Universal Robots PolyScope program: 6 novembre.urp

Program 6 novembre (installation=default directory=/programs createdIn=3.15.8.106339 lastSavedIn=3.15.8.106339 robotSerialNumber=2023330214)
Calibrated DH parameters: a=[-0.000161, -0.243516, -0.175941, 0.000055, -0.000127, 0]; d=[0.151869, -0.926342, 57.568096, -56.529557, 0.085345, 0.082309]; alpha=[1.571543, -0.007517, 0.002128, 1.570286, -1.573097, 0]; deltaTheta=[0.000048, 0.028487, 0.571925, -0.600676, 0.000055, 0.000013]
BeforeStart
  conta := 0
Robot Program (runOnlyOnce=false)
  Loop Counting (count=5) loopVariable(name=Loop_1)
    MoveJ speed 60 deg/s, acceleration 80 deg/s^2 (useActiveTCP=true)
      Waypoint partenza: motionParameters(jointSpeed=6.283185 jointAcceleration=6.283185 cartesianSpeed=0.25 cartesianAcceleration=1.2); TCP in base x=295.823 y=29.54 z=245.993 mm, rx=-1.6446 ry=2.6015 rz=0.0088 rad; joints [31.55, -87.588, -89.18, -89.432, 90.433, 57.296] deg; flange x=307.635 y=60.145 z=330.959 mm, rx=-1.6446 ry=2.6015 rz=0.0088 rad
      Pallet pattern(dimensionality=Square firstAxisCount=2 secondAxisCount=2 thirdAxisCount=5 motionType=MoveL speed=0.25 acceleration=1.2 useActiveTCP=true, counterVariable(name=cnt_1, initializeExpression=0), patternPoseVariable(name=pose_1), feature=Base, children(Waypoint(type=Fixed name=Corner1_2, position(joints=1.7071903944015503, -2.0363944212542933, -1.974642578755514, -0.7177489439593714, 1.586946964263916, 1.8594038486480713 pose=0.05591609202787988, 0.3042326877636343, 0.04062971376229775, 2.037561659965045, -2.3576852381341817, 0.00967614852521311), poseInFeatureCoordinates=[0.055916, 0.304233, 0.04063, 2.037562, -2.357685, 0.009676], outputFlangePose=[0.062603, 0.343098, 0.122727, 2.037562, -2.357685, 0.009676]), Waypoint(type=Fixed name=Corner2_2, position(joints=1.3555443286895752, -2.164708439503805, -1.7350428740130823, -0.8342025915728968, 1.5785411596298218, 1.5071099996566772 pose=0.18014491122547477, 0.3042332340391118, 0.04060207246304333, 2.037508402011708, -2.357604882143758, 0.009722233499361176), poseInFeatureCoordinates=[0.180145, 0.304233, 0.040602, 2.037508, -2.357605, 0.009722], outputFlangePose=[0.186836, 0.343105, 0.122696, 2.037508, -2.357605, 0.009722]), Waypoint(type=Fixed name=Corner3_2, position(joints=1.2638148069381714, -1.8657797018634241, -2.2631152311908167, -0.6058977285968226, 1.5782291889190674, 1.4168099164962769 pose=0.18015284222828584, 0.1875657559943738, 0.04061133384541858, 2.03742066799229, -2.3576919944708794, 0.009735192963967047), poseInFeatureCoordinates=[0.180153, 0.187566, 0.040611, 2.037421, -2.357692, 0.009735], outputFlangePose=[0.186846, 0.226438, 0.122705, 2.037421, -2.357692, 0.009735]), Waypoint(type=Fixed name=Corner4_2, position(joints=1.8628913164138794, -1.6507962385760706, -2.576595131550924, -0.49827701250185186, 1.5922470092773438, 2.016301393508911 pose=0.03904266180606819, 0.18759146961099127, 0.040612373225184156, 2.0374934541390837, -2.3578468661229373, 0.009639408672472292), poseInFeatureCoordinates=[0.039043, 0.187591, 0.040612, 2.037493, -2.357847, 0.009639], outputFlangePose=[0.04573, 0.22645, 0.122713, 2.037493, -2.357847, 0.009639]))); actionSequence(name=PalletSequence motionType=MoveL speed=0.25 acceleration=1.2 useActiveTCP=true, anchorWaypoint(type=Fixed name=PatternPoint_2), feature=Base, children(Waypoint(type=Fixed name=Approach_2), Waypoint=PatternPoint_2, Set(type=Undefined), Wait(type=Undefined), Waypoint(type=Fixed name=Exit_2)))
        Pattern -> pattern
        AnchoredSequence -> PalletSequence
      Pallet pattern(dimensionality=Box firstAxisCount=2 secondAxisCount=2 thirdAxisCount=2 motionType=MoveL speed=2 acceleration=2 useActiveTCP=true, counterVariable(name=cnt_2, initializeExpression=0), patternPoseVariable(name=pose_2), feature=Base, children(Waypoint(type=Fixed name=Corner1_1, position(joints=1.5661438703536987, -2.322768513356344, -1.645829979573385, -0.6583693663226526, 1.5955449342727661, 0.8307483792304993 pose=0.13254062465471933, 0.3819871783574357, 0.01202495287692959, -2.815561845639961, 1.238537976676179, 0.09161537053473316), poseInFeatureCoordinates=[0.132541, 0.381987, 0.012025, -2.815562, 1.238538, 0.091615], outputFlangePose=[0.109614, 0.402639, 0.097717, -2.815562, 1.238538, 0.091615]), Waypoint(type=Fixed name=Corner2_1, position(joints=2.069969415664673, -2.30833083788027, -1.6788514296161097, -0.6362593809710901, 1.552017092704773, 1.33286714553833 pose=-0.06981415651235434, 0.3820034575878895, 0.012055526427345212, -2.8153862369095832, 1.2386705000643832, 0.09160329857243932), poseInFeatureCoordinates=[-0.069814, 0.382003, 0.012056, -2.815386, 1.238671, 0.091603], outputFlangePose=[-0.092742, 0.40265, 0.097749, -2.815386, 1.238671, 0.091603]), Waypoint(type=Fixed name=Corner3_1, position(joints=2.1814701557159424, -2.1197527090655726, -2.091782871876852, -0.4142039457904261, 1.5434199571609497, 1.4452728033065796 pose=-0.06985309927787037, 0.3076010722744215, 0.012025167135886666, -2.81546452850973, 1.2386318532493505, 0.09155135403268563), poseInFeatureCoordinates=[-0.069853, 0.307601, 0.012025, -2.815465, 1.238632, 0.091551], outputFlangePose=[-0.092783, 0.328252, 0.097717, -2.815465, 1.238632, 0.091551]), Waypoint(type=Fixed name=Corner4_1, position(joints=1.6141332387924194, -2.1172483603106897, -2.0820215384112757, -0.42622596422304326, 1.5924631357192993, 0.8800121545791626 pose=0.11696996682890427, 0.30762812058442696, 0.013640332231584604, -2.8154065555165144, 1.2384555292847788, 0.09165857290291884), poseInFeatureCoordinates=[0.11697, 0.307628, 0.01364, -2.815407, 1.238456, 0.091659], outputFlangePose=[0.09404, 0.328265, 0.099335, -2.815407, 1.238456, 0.091659]), Waypoint(type=Fixed name=Corner5_1, position(joints=1.5661195516586304, -2.2069433371173304, -1.6129887739764612, -0.8070271650897425, 1.5962883234024048, 0.8310835361480713 pose=0.13254505804894007, 0.3819913606874764, 0.05326265409589624, -2.8155296229078335, 1.2386440785686519, 0.09166160286875408), poseInFeatureCoordinates=[0.132545, 0.381991, 0.053263, -2.81553, 1.238644, 0.091662], outputFlangePose=[0.109623, 0.402645, 0.138956, -2.81553, 1.238644, 0.091662]), Waypoint(type=Fixed name=Corner6_1, position(joints=1.8421919345855713, -1.758475128804342, -2.226459805165426, -0.6699078718768519, 1.5725816488265991, 1.669399619102478 pose=0.03699638008789556, 0.2645854558919123, 0.06973987779796274, -2.3891578310447525, 1.993011190932662, 0.07230867192476798), poseInFeatureCoordinates=[0.036996, 0.264585, 0.06974, -2.389158, 1.993011, 0.072309], outputFlangePose=[0.031683, 0.297078, 0.154659, -2.389158, 1.993011, 0.072309]), Waypoint(type=Fixed name=Corner7_1, position(joints=2.1814942359924316, -1.9579713980304163, -2.053600613270895, -0.6142085234271448, 1.5447266101837158, 1.4454758167266846 pose=-0.06988329350081754, 0.3075806044495836, 0.053988135413453, -2.8155694251031185, 1.238588640015896, 0.09155601460152367), poseInFeatureCoordinates=[-0.069883, 0.307581, 0.053988, -2.815569, 1.238589, 0.091556], outputFlangePose=[-0.092811, 0.328236, 0.139679, -2.815569, 1.238589, 0.091556]), Waypoint(type=Fixed name=Corner8_1, position(joints=1.6140732765197754, -1.9632557074176233, -2.0447023550616663, -0.6174734274493616, 1.5936022996902466, 0.8802626729011536 pose=0.11697436518505036, 0.30764425213376984, 0.05402597240678174, -2.8152865555920723, 1.2385633191985477, 0.0916434361586064), poseInFeatureCoordinates=[0.116974, 0.307644, 0.054026, -2.815287, 1.238563, 0.091643], outputFlangePose=[0.094044, 0.328279, 0.139721, -2.815287, 1.238563, 0.091643]))); actionSequence(name=PalletSequence motionType=MoveL speed=2 acceleration=2 useActiveTCP=true, anchorWaypoint(type=Fixed name=PatternPoint_1, position(joints=1.5661075115203857, -2.3227208296405237, -1.6458538214312952, -0.6583455244647425, 1.5955688953399658, 0.8307603597640991 pose=0.13255022991976123, 0.3819850223950209, 0.012039257013669744, -2.8154995143954062, 1.2385888289909233, 0.09167611634166095), poseInFeatureCoordinates=[0.13255, 0.381985, 0.012039, -2.8155, 1.238589, 0.091676], outputFlangePose=[0.109627, 0.402634, 0.097733, -2.8155, 1.238589, 0.091676]), feature=Base, children(Waypoint(type=Fixed name=Approach_1, position(joints=1.5661195516586304, -2.1142290274249476, -1.5500968138324183, -0.9625776449786585, 1.596911907196045, 0.8311670422554016 pose=0.13255691953557736, 0.38198130637054345, 0.09323890177774338, -2.8155039252593643, 1.2386177840645376, 0.09174743687930356), poseInFeatureCoordinates=[0.132557, 0.381981, 0.093239, -2.815504, 1.238618, 0.091747], outputFlangePose=[0.109638, 0.40263, 0.178934, -2.815504, 1.238618, 0.091747]), Waypoint=PatternPoint_1, Assignment(valueSource=Expression, variable=conta, expression=conta+1), Popup(type=Message haltProgram=false message=oggetto posato inputType=Variable, variable=conta), Wait(type=Sleep, waitTime=2), Waypoint(type=Fixed name=Exit_1, position(joints=1.566071629524231, -2.1142171064959925, -1.5500367323504847, -0.9625890890704554, 1.5968759059906006, 0.8311071395874023 pose=0.1325829007796406, 0.38199128837101787, 0.09325883660014188, -2.81544429941611, 1.2385730377346045, 0.09172694314242495), poseInFeatureCoordinates=[0.132583, 0.381991, 0.093259, -2.815444, 1.238573, 0.091727], outputFlangePose=[0.10966, 0.402635, 0.178954, -2.815444, 1.238573, 0.091727])))
        Pattern -> pattern
        AnchoredSequence -> PalletSequence
